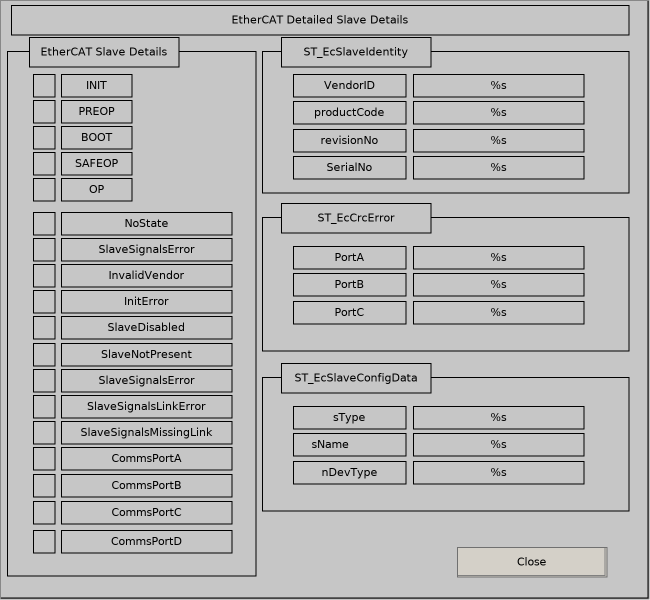
VISUALIZATION diagEtherCATSlaveDetail  // 650x600
VAR_IN_OUT
	dataValues:typeEtherCATIndicator;
END_VAR
    Rectangle (0,0 648x598)
    Rectangle (262,51 367x142)
    Rectangle (7,51 249x525)
    Rectangle (33,74 22x23)
    Rectangle (61,74 71x23), "INIT"
    Rectangle (33,100 22x23)
    Rectangle (61,100 71x23), "PREOP"
    Rectangle (33,126 22x23)
    Rectangle (61,126 71x23), "BOOT"
    Rectangle (33,152 22x23)
    Rectangle (61,152 71x23), "SAFEOP"
    Rectangle (33,178 22x23)
    Rectangle (61,178 71x23), "OP"
    Rectangle (33,212 22x23)
    Rectangle (61,212 171x23), "NoState"
    Rectangle (33,238 22x23)
    Rectangle (61,238 171x23), "SlaveSignalsError"
    Rectangle (33,264 22x23)
    Rectangle (61,264 171x23), "InvalidVendor"
    Rectangle (33,290 22x23)
    Rectangle (61,290 171x23), "InitError"
    Rectangle (33,316 22x23)
    Rectangle (61,316 171x23), "SlaveDisabled"
    Rectangle (33,343 22x23)
    Rectangle (61,343 171x23), "SlaveNotPresent"
    Rectangle (33,369 22x23)
    Rectangle (61,369 171x23), "SlaveSignalsError"
    Rectangle (33,395 22x23)
    Rectangle (61,395 171x23), "SlaveSignalsLinkError"
    Rectangle (33,421 22x23)
    Rectangle (61,421 171x23), "SlaveSignalsMissingLink"
    Rectangle (33,447 22x23)
    Rectangle (61,447 171x23), "CommsPortA"
    Rectangle (33,474 22x23)
    Rectangle (61,474 171x23), "CommsPortB"
    Rectangle (33,501 22x23)
    Rectangle (61,501 171x23), "CommsPortC"
    Rectangle (33,530 22x23)
    Rectangle (61,530 171x23), "CommsPortD"
    Rectangle (29,37 150x30), "EtherCAT Slave Details"
    Rectangle (293,74 113x23), "VendorID"
    Rectangle (413,74 171x23), "%s", text variable: dataValues.ConfigData.stSlaveIdentity.vendorId
    Rectangle (413,101 171x23), "%s", text variable: dataValues.ConfigData.stSlaveIdentity.productCode
    Rectangle (293,101 113x23), "productCode"
    Rectangle (293,129 113x23), "revisionNo"
    Rectangle (413,129 171x23), "%s", text variable: dataValues.ConfigData.stSlaveIdentity.revisionNo
    Rectangle (413,156 171x23), "%s", text variable: dataValues.ConfigData.stSlaveIdentity.serialNo
    Rectangle (293,156 113x23), "SerialNo"
    Rectangle (281,37 150x30), "ST_EcSlaveIdentity"
    Rectangle (262,217 367x134)
    Rectangle (293,246 113x23), "PortA"
    Rectangle (413,246 171x23), "%s", text variable: dataValues.crcCount.portA
    Rectangle (413,273 171x23), "%s", text variable: dataValues.crcCount.portB
    Rectangle (293,273 113x23), "PortB"
    Rectangle (293,301 113x23), "PortC"
    Rectangle (413,301 171x23), "%s", text variable: dataValues.crcCount.portC
    Rectangle (281,203 150x30), "ST_EcCrcError"
    Rectangle (262,377 367x134)
    Rectangle (293,406 113x23), "sType"
    Rectangle (413,406 171x23), "%s", text variable: dataValues.ConfigData.sType
    Rectangle (413,433 171x23), "%s", text variable: dataValues.ConfigData.sName
    Rectangle (293,433 113x23), "sName"
    Rectangle (293,461 113x23), "nDevType"
    Rectangle (413,461 171x23), "%s", text variable: dataValues.ConfigData.nDevType
    Rectangle (281,363 150x30), "ST_EcSlaveConfigData"
    Button (457,547 150x30), "Close"
        OnMouseClick: CloseDialog Dialog=diagEtherCATSlaveDetail, Result=None, NumpadKeypadSet=True
    Rectangle (11,5 618x30), "EtherCAT Detailed Slave Details"
END_VISUALIZATION

(* stored: Version 1.1.0.1, ProductVersion 3.1.4024.12
   Visu diagEtherCATSlaveDetail: Id {0e5479e1-51c5-4cc7-a392-006154e867e4} *)
